{attribute addProperty BoxType "ELX1052-0000-0016"}
{attribute addProperty Id "ChannelAT %I*ARRAY[0..2] OF Channel_E18390663240WcStateAT %I*WcState_98A4DF7520.250InfoDataAT %I*InfoData_192954DE1620"}
{attribute addProperty CRC "795057235"}
{attribute addProperty SizeInBites "50"}
{attribute addProperty SizeInBytes "6.25"}
TYPE ELX1052_F21EA95A :
STRUCT
	{attribute addProperty Name "Channel"}
	Channel : ARRAY[0..2] OF Channel_E1839066;
	{attribute addProperty Name "WcState"}
	WcState : WcState_98A4DF75;
	{attribute addProperty Name "InfoData"}
	InfoData : InfoData_192954DE;
END_STRUCT
END_TYPE

(* stored: Version 1.2.0.0, ProductVersion 3.1.4024.9
   DUT ELX1052_F21EA95A: Id {d8c15e54-e5df-4378-ab50-05afdb6bfc17} *)
